(* IEC 61131-3 sources: ae-trafficlight/src, 7 files *)

(* ---- StateGreen.st ---- *)
USING Simatic.Ax.Stateframework;
USING Simatic.Ax.SimpleControlModules;

NAMESPACE ApplicationStateFramwerok
    CLASS StateGreen EXTENDS State1Transition

        VAR PUBLIC
            LightStack : REF_TO LightStackRdYeGnBl;
        END_VAR

        METHOD PUBLIC OVERRIDE OnEntry
            LightStack^.SwitchOn(Colors#Green);
        END_METHOD

        METHOD PUBLIC OVERRIDE OnExit
            LightStack^.SwitchOff(Colors#Green);
        END_METHOD

        METHOD PUBLIC OVERRIDE Action
            ;
        END_METHOD

    END_CLASS
END_NAMESPACE

(* ---- StateInit.st ---- *)
USING Simatic.Ax.Stateframework;
USING Simatic.Ax.SimpleControlModules;

NAMESPACE ApplicationStateFramwerok
    CLASS StateInit EXTENDS State1Transition

        VAR  PUBLIC
            LightStack : REF_TO LightStackRdYeGnBl;
        END_VAR

        METHOD PUBLIC OVERRIDE OnEntry
            LightStack^.SwitchOn(Colors#Red);
            LightStack^.SwitchOn(Colors#Yellow);
            LightStack^.SwitchOn(Colors#Green);
        END_METHOD

        METHOD PUBLIC OVERRIDE OnExit
            LightStack^.SwitchOff(Colors#Red);
            LightStack^.SwitchOff(Colors#Yellow);
            LightStack^.SwitchOff(Colors#Green);
        END_METHOD

        METHOD PUBLIC OVERRIDE Action
            ;
        END_METHOD

    END_CLASS
END_NAMESPACE

(* ---- StateRed.st ---- *)
USING Simatic.Ax.Stateframework;
USING Simatic.Ax.SimpleControlModules;

NAMESPACE ApplicationStateFramwerok
    CLASS StateRed EXTENDS State1Transition

        VAR  PUBLIC
            LightStack : REF_TO LightStackRdYeGnBl;
        END_VAR

        METHOD PUBLIC OVERRIDE OnEntry
            LightStack^.SwitchOn(Colors#Red);
        END_METHOD

        METHOD PUBLIC OVERRIDE OnExit
            LightStack^.SwitchOff(Colors#Red);
        END_METHOD

        METHOD PUBLIC OVERRIDE Action
            ;
        END_METHOD

    END_CLASS
END_NAMESPACE

(* ---- StateRedYellow.st ---- *)
USING Simatic.Ax.Stateframework;
USING Simatic.Ax.SimpleControlModules;

NAMESPACE ApplicationStateFramwerok
    CLASS StateRedYellow EXTENDS State1Transition

        VAR  PUBLIC
            LightStack : REF_TO LightStackRdYeGnBl;
        END_VAR

        METHOD PUBLIC OVERRIDE OnEntry
            LightStack^.SwitchOn(Colors#Red);
            LightStack^.SwitchOn(Colors#Yellow);
        END_METHOD

        METHOD PUBLIC OVERRIDE OnExit
            LightStack^.SwitchOff(Colors#Red);
            LightStack^.SwitchOff(Colors#Yellow);
        END_METHOD

        METHOD PUBLIC OVERRIDE Action
            ;
        END_METHOD

    END_CLASS
END_NAMESPACE

(* ---- StateYellow.st ---- *)
USING Simatic.Ax.Stateframework;
USING Simatic.Ax.SimpleControlModules;

NAMESPACE ApplicationStateFramwerok
    CLASS StateYellow EXTENDS State1Transition

        VAR  PUBLIC
            LightStack : REF_TO LightStackRdYeGnBl;
        END_VAR

        METHOD PUBLIC OVERRIDE OnEntry
            LightStack^.SwitchOn(Colors#Yellow);
        END_METHOD

        METHOD PUBLIC OVERRIDE OnExit
            LightStack^.SwitchOff(Colors#Yellow);
        END_METHOD

        METHOD PUBLIC OVERRIDE Action
            ;
        END_METHOD

    END_CLASS
END_NAMESPACE

(* ---- Configuration.st ---- *)
USING Simatic.Ax.StateFramework;
USING Simatic.Ax.IO.Output;
USING Simatic.Ax.SimpleControlModules;
USING ApplicationStateFramwerok;
CONFIGURATION MyConfiguration
    TASK Main(Priority := 1);

    PROGRAM P1 WITH Main: MainProgram;

    // Configuring IO tags
    VAR_GLOBAL
        QRd AT %Q0.0 : BOOL;
        QYe AT %Q0.1 : BOOL;
        QGn AT %Q0.2 : BOOL;
    END_VAR

    // Configuring the global equipment
    VAR_GLOBAL
        TrafficLight : LightStackRdYeGnBl := (QRed := QRed, QYellow := QYellow, QGreen := QGreen);
        QRed : BinOutput;
        QYellow : BinOutput;
        QGreen : BinOutput;
        ActiveStateName : STRING;
    END_VAR

    // Configuring the state machine
    VAR_GLOBAL
        StateController : StateController := (InitialState := InitState);
        // Initial State
        InitGuard : TRUEGUARD; //TimeoutGuard := (Timeout := T#3000ms);
        Init2Red : Transition := (Guard := InitGuard, NextState := RedState);
        InitState : StateInit := (StateName := 'Init', Transition1 := Init2Red, LightStack := REF(TrafficLight));

        // State Red
        RedGuard : TimeoutGuard := (Timeout := T#1500ms);
        Red2RedYellow : Transition := (Guard := RedGuard, NextState := RedYellowState);
        RedState : StateRed := (StateName := 'Red', Transition1 := Red2RedYellow, LightStack := REF(TrafficLight));

        // State RedYellow
        RedYellowGuard : TimeoutGuard := (Timeout := T#1500ms);
        RedYellowToGreen : Transition := (Guard := RedYellowGuard, NextState := GreenState);
        RedYellowState : StateRedYellow := (StateName := 'RedYellow', Transition1 := RedYellowToGreen, LightStack := REF(TrafficLight));

        // State Green
        GreenGuard : TimeoutGuard := (Timeout := T#1500ms);
        Green2Yellow : Transition := (Guard := GreenGuard, NextState := YellowState);
        GreenState : StateGreen := (StateName := 'Green', Transition1 := Green2Yellow, LightStack := REF(TrafficLight));

        // State Yellow
        YellowGuard : TimeoutGuard := (Timeout := T#1500ms);
        Yellow2Count : Transition := (Guard := YellowGuard, NextState := CycleCountState);
        YellowState : StateYellow := (StateName := 'Yellow', Transition1 := Yellow2Count, LightStack := REF(TrafficLight));

        // Check Cycles
        CycleCountGuard : CountGuard := (count := LINT#5);
        CycleCountAlwaysTrueGuard : TrueGuard;
        CycleCountToInit : Transition := (Guard := CycleCountGuard, NextState := InitState);
        CycleCountToRed: Transition := (Guard := CycleCountAlwaysTrueGuard, NextState := RedState);
        CycleCountState : State2Transition := (StateID := 6, Transition1 := CycleCountToInit, transition2 := CycleCountToRed);

    END_VAR
END_CONFIGURATION

(* ---- MainProgram.st ---- *)
USING Simatic.Ax.StateFramework;
USING Simatic.Ax.IO.Output;
USING Simatic.Ax.SimpleControlModules;

PROGRAM MainProgram
    VAR_EXTERNAL
        StateController : StateController;
        TrafficLight : LightStackRdYeGnBl;

        QRd : BOOL;
        QYe : BOOL;
        QGn : BOOL;
        ActiveStateName : STRING;

    END_VAR

    StateController.Execute();
    QRd := TrafficLight.GetState(Colors#Red);
    QYe := TrafficLight.GetState(Colors#Yellow);
    QGn := TrafficLight.GetState(Colors#Green);
    ActiveStateName := StateController.GetActiveStateName();
END_PROGRAM

// test 7
